TYPE CUBaseSettings EXTENDS TcoCore.TcoStruct : STRUCT
    DeafultCycleTime : TIME;
    WarningCycleTime : TIME;
    ErrorCycleTime : TIME;
    SaveEnergyTime : TIME;
    AnyRecurringFailure : UINT;
    SameRecurringFailure : UINT;
END_STRUCT
END_TYPE

(* stored: Version 1.1.0.1
   DUT CUBaseSettings: Id {9173d902-7cba-0c0b-1d10-4c6f12b76cb5} *)
